SYSTEM TestDataType
  (* Version 1.0, 2024-01-14, ADMIN *)
  APPLICATION TestDataTypeApp
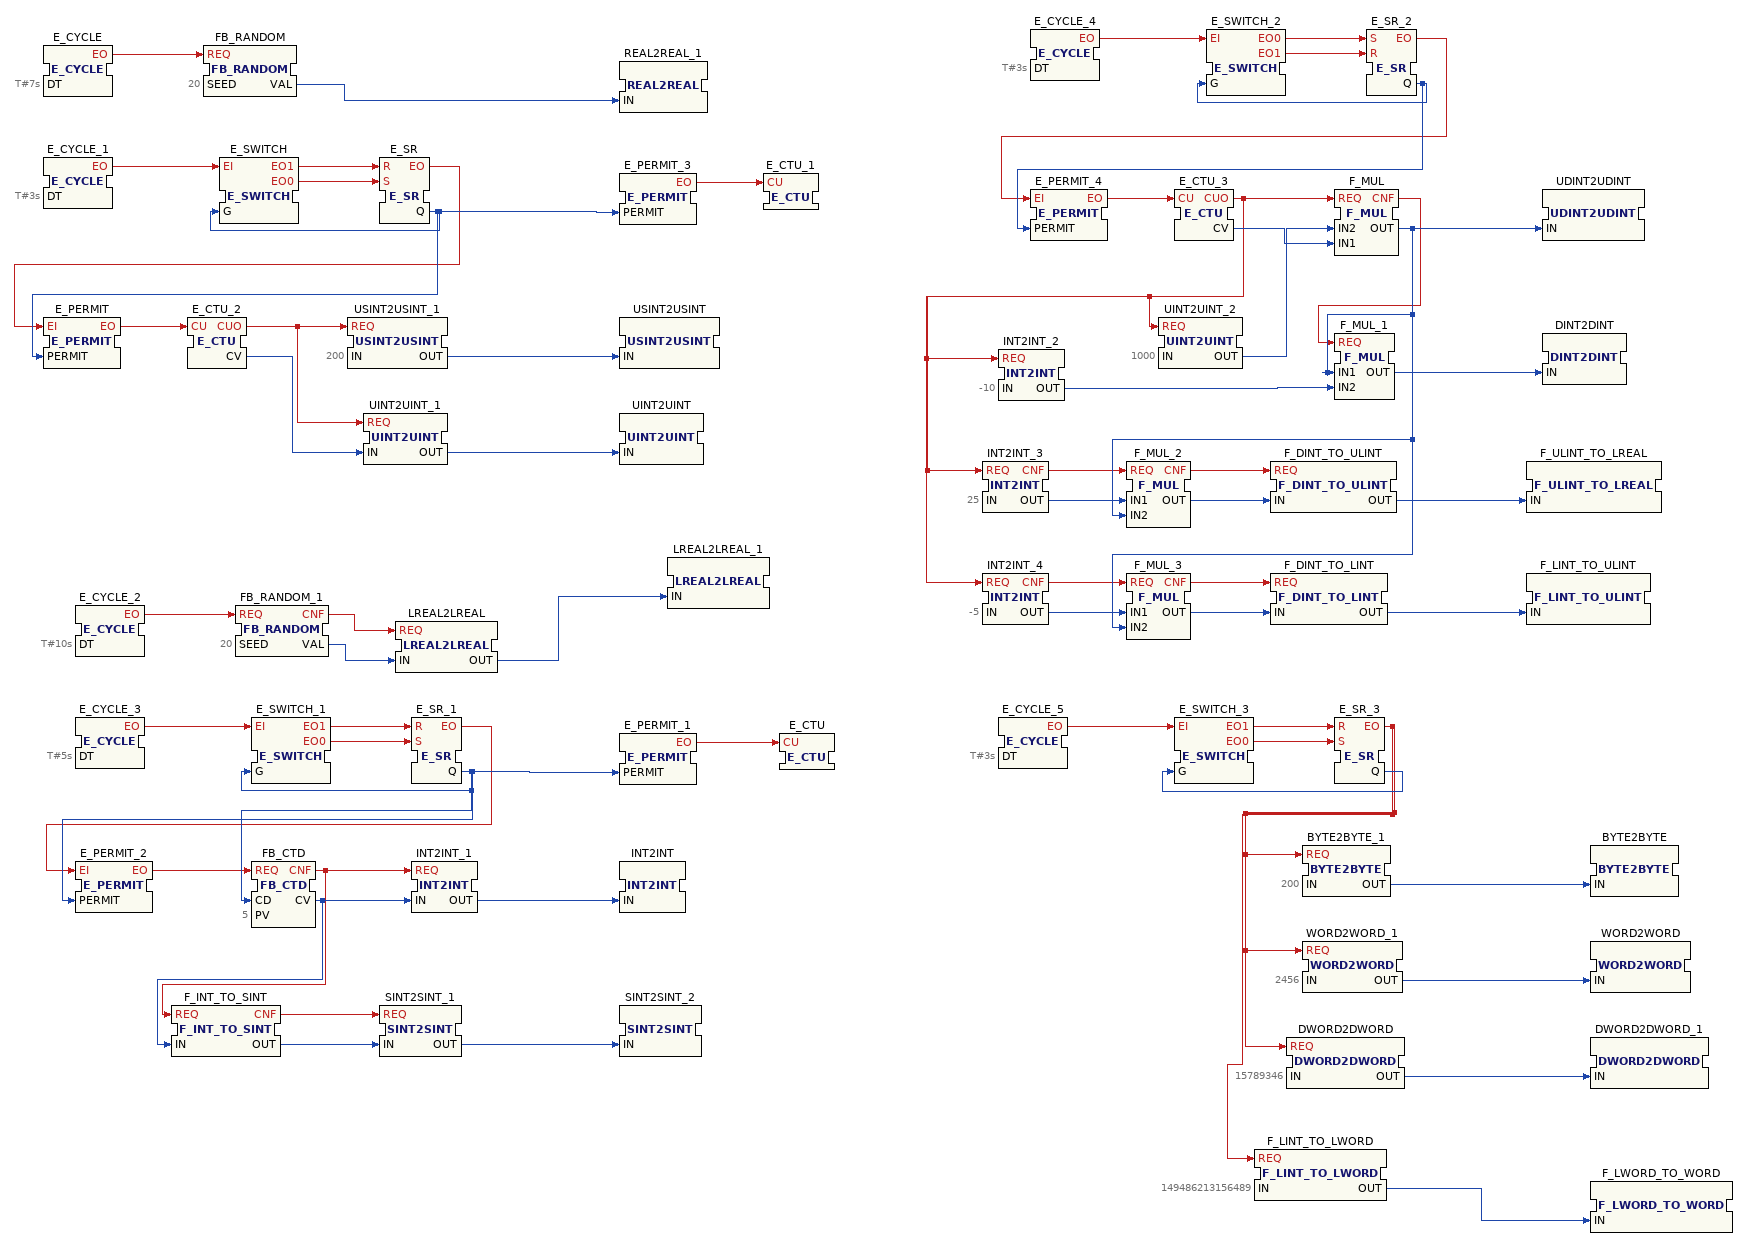
    FBS
      E_CYCLE : E_CYCLE(DT := T#7s);
      FB_RANDOM : FB_RANDOM(SEED := 20);
      E_CYCLE_1 : E_CYCLE(DT := T#3s);
      E_SWITCH : E_SWITCH;
      E_SR : E_SR;
      E_PERMIT : E_PERMIT;
      E_PERMIT_1 : E_PERMIT;
      E_CTU : E_CTU;
      E_CYCLE_2 : E_CYCLE(DT := T#10s);
      FB_RANDOM_1 : FB_RANDOM(SEED := 20);
      E_CYCLE_3 : E_CYCLE(DT := T#5s);
      E_SWITCH_1 : E_SWITCH;
      E_SR_1 : E_SR;
      E_PERMIT_2 : E_PERMIT;
      REAL2REAL_1 : REAL2REAL;
      E_PERMIT_3 : E_PERMIT;
      E_CTU_1 : E_CTU;
      UINT2UINT : UINT2UINT;
      INT2INT : INT2INT;
      SINT2SINT_1 : SINT2SINT;
      USINT2USINT : USINT2USINT;
      E_CTU_2 : E_CTU;
      UINT2UINT_1 : UINT2UINT;
      SINT2SINT_2 : SINT2SINT;
      INT2INT_1 : INT2INT;
      USINT2USINT_1 : USINT2USINT(IN := 200);
      LREAL2LREAL : LREAL2LREAL;
      LREAL2LREAL_1 : LREAL2LREAL;
      UDINT2UDINT : UDINT2UDINT;
      DINT2DINT : DINT2DINT;
      F_MUL : F_MUL;
      UINT2UINT_2 : UINT2UINT(IN := 1000);
      FB_CTD : FB_CTD(PV := 5);
      F_INT_TO_SINT : F_INT_TO_SINT;
      E_CYCLE_4 : E_CYCLE(DT := T#3s);
      E_SWITCH_2 : E_SWITCH;
      E_SR_2 : E_SR;
      E_PERMIT_4 : E_PERMIT;
      E_CTU_3 : E_CTU;
      F_MUL_1 : F_MUL;
      INT2INT_2 : INT2INT(IN := -10);
      BYTE2BYTE : BYTE2BYTE;
      WORD2WORD : WORD2WORD;
      F_DINT_TO_LINT : F_DINT_TO_LINT;
      F_LINT_TO_ULINT : F_LINT_TO_ULINT;
      F_DINT_TO_ULINT : F_DINT_TO_ULINT;
      INT2INT_3 : INT2INT(IN := 25);
      F_MUL_2 : F_MUL;
      F_ULINT_TO_LREAL : F_ULINT_TO_LREAL;
      INT2INT_4 : INT2INT(IN := -5);
      F_MUL_3 : F_MUL;
      E_SWITCH_3 : E_SWITCH;
      E_SR_3 : E_SR;
      E_CYCLE_5 : E_CYCLE(DT := T#3s);
      BYTE2BYTE_1 : BYTE2BYTE(IN := 200);
      DWORD2DWORD : DWORD2DWORD(IN := 15789346);
      WORD2WORD_1 : WORD2WORD(IN := 2456);
      DWORD2DWORD_1 : DWORD2DWORD;
      F_LWORD_TO_WORD : F_LWORD_TO_WORD;
      F_LINT_TO_LWORD : F_LINT_TO_LWORD(IN := 149486213156489);
    END_FBS
    EVENT_CONNECTIONS
      E_CYCLE.EO TO FB_RANDOM.REQ;
      E_SWITCH.EO1 TO E_SR.R;
      E_SWITCH.EO0 TO E_SR.S;
      E_SR.EO TO E_PERMIT.EI;
      E_CYCLE_1.EO TO E_SWITCH.EI;
      E_PERMIT_1.EO TO E_CTU.CU;
      E_PERMIT_3.EO TO E_CTU_1.CU;
      E_SR_1.EO TO E_PERMIT_2.EI;
      E_CYCLE_2.EO TO FB_RANDOM_1.REQ;
      E_SWITCH_1.EO1 TO E_SR_1.R;
      E_CYCLE_3.EO TO E_SWITCH_1.EI;
      E_SWITCH_1.EO0 TO E_SR_1.S;
      E_PERMIT.EO TO E_CTU_2.CU;
      E_CTU_2.CUO TO UINT2UINT_1.REQ;
      E_CTU_2.CUO TO USINT2USINT_1.REQ;
      FB_RANDOM_1.CNF TO LREAL2LREAL.REQ;
      E_PERMIT_2.EO TO FB_CTD.REQ;
      FB_CTD.CNF TO INT2INT_1.REQ;
      F_INT_TO_SINT.CNF TO SINT2SINT_1.REQ;
      FB_CTD.CNF TO F_INT_TO_SINT.REQ;
      E_PERMIT_4.EO TO E_CTU_3.CU;
      E_CYCLE_4.EO TO E_SWITCH_2.EI;
      E_SWITCH_2.EO0 TO E_SR_2.S;
      E_SR_2.EO TO E_PERMIT_4.EI;
      E_SWITCH_2.EO1 TO E_SR_2.R;
      E_CTU_3.CUO TO F_MUL.REQ;
      E_CTU_3.CUO TO UINT2UINT_2.REQ;
      E_CTU_3.CUO TO INT2INT_2.REQ;
      F_MUL.CNF TO F_MUL_1.REQ;
      E_CTU_3.CUO TO INT2INT_3.REQ;
      INT2INT_3.CNF TO F_MUL_2.REQ;
      F_MUL_2.CNF TO F_DINT_TO_ULINT.REQ;
      F_MUL_3.CNF TO F_DINT_TO_LINT.REQ;
      E_CTU_3.CUO TO INT2INT_4.REQ;
      INT2INT_4.CNF TO F_MUL_3.REQ;
      E_CYCLE_5.EO TO E_SWITCH_3.EI;
      E_SWITCH_3.EO1 TO E_SR_3.R;
      E_SWITCH_3.EO0 TO E_SR_3.S;
      E_SR_3.EO TO BYTE2BYTE_1.REQ;
      E_SR_3.EO TO WORD2WORD_1.REQ;
      E_SR_3.EO TO DWORD2DWORD.REQ;
      E_SR_3.EO TO F_LINT_TO_LWORD.REQ;
    END_CONNECTIONS
    DATA_CONNECTIONS
      E_SR.Q TO E_SWITCH.G;
      E_SR.Q TO E_PERMIT.PERMIT;
      E_SR_1.Q TO E_SWITCH_1.G;
      E_SR_1.Q TO E_PERMIT_2.PERMIT;
      E_SR.Q TO E_PERMIT_3.PERMIT;
      E_SR_1.Q TO E_PERMIT_1.PERMIT;
      FB_RANDOM.VAL TO REAL2REAL_1.IN;
      E_CTU_2.CV TO UINT2UINT_1.IN;
      INT2INT_1.OUT TO INT2INT.IN;
      SINT2SINT_1.OUT TO SINT2SINT_2.IN;
      USINT2USINT_1.OUT TO USINT2USINT.IN;
      UINT2UINT_1.OUT TO UINT2UINT.IN;
      FB_RANDOM_1.VAL TO LREAL2LREAL.IN;
      LREAL2LREAL.OUT TO LREAL2LREAL_1.IN;
      FB_CTD.CV TO INT2INT_1.IN;
      F_INT_TO_SINT.OUT TO SINT2SINT_1.IN;
      FB_CTD.CV TO F_INT_TO_SINT.IN;
      E_SR_2.Q TO E_PERMIT_4.PERMIT;
      E_SR_2.Q TO E_SWITCH_2.G;
      UINT2UINT_2.OUT TO F_MUL.IN2;
      E_CTU_3.CV TO F_MUL.IN1;
      F_MUL.OUT TO F_MUL_1.IN1;
      INT2INT_2.OUT TO F_MUL_1.IN2;
      F_MUL.OUT TO UDINT2UDINT.IN;
      F_MUL_1.OUT TO DINT2DINT.IN;
      E_SR_1.Q TO FB_CTD.CD;
      INT2INT_3.OUT TO F_MUL_2.IN1;
      F_MUL.OUT TO F_MUL_2.IN2;
      F_MUL_2.OUT TO F_DINT_TO_ULINT.IN;
      F_DINT_TO_LINT.OUT TO F_LINT_TO_ULINT.IN;
      F_DINT_TO_ULINT.OUT TO F_ULINT_TO_LREAL.IN;
      INT2INT_4.OUT TO F_MUL_3.IN1;
      F_MUL.OUT TO F_MUL_3.IN2;
      F_MUL_3.OUT TO F_DINT_TO_LINT.IN;
      E_SR_3.Q TO E_SWITCH_3.G;
      BYTE2BYTE_1.OUT TO BYTE2BYTE.IN;
      WORD2WORD_1.OUT TO WORD2WORD.IN;
      DWORD2DWORD.OUT TO DWORD2DWORD_1.IN;
      F_LINT_TO_LWORD.OUT TO F_LWORD_TO_WORD.IN;
    END_CONNECTIONS
  END_APPLICATION
  DEVICE BeagleBoneBlack : BeagleBoneBlack(MGR_ID := "localhost:61500")
    {SET_ATTRIBUTE(Profile, HOLOBLOC)} (* device profile *)
    RESOURCE EMB_RES : EMB_RES
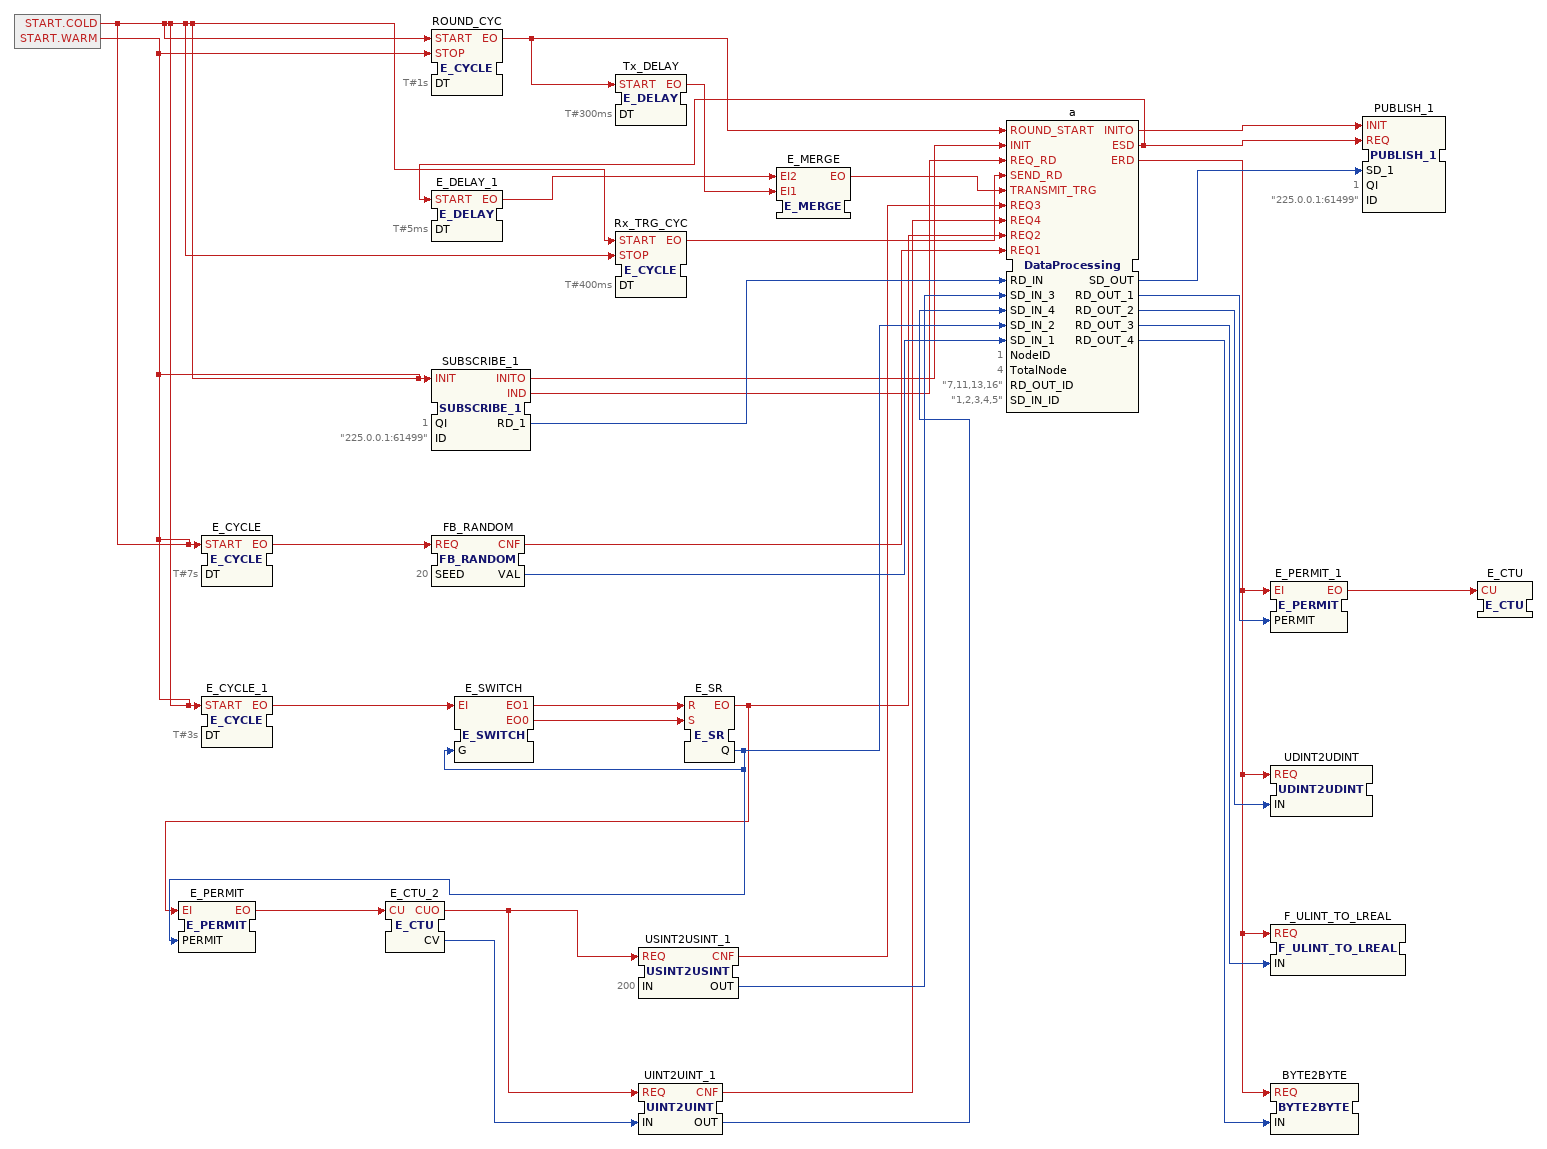
      FBS
        a : DataProcessing(NodeID := 1, TotalNode := 4, RD_OUT_ID := "7,11,13,16", SD_IN_ID := "1,2,3,4,5");
        Rx_TRG_CYC : E_CYCLE(DT := T#400ms);
        PUBLISH_1 : PUBLISH_1(QI := 1, ID := "225.0.0.1:61499");
        E_DELAY_1 : E_DELAY(DT := T#5ms);
        SUBSCRIBE_1 : SUBSCRIBE_1(QI := 1, ID := "225.0.0.1:61499");
        E_MERGE : E_MERGE;
        Tx_DELAY : E_DELAY(DT := T#300ms);
        ROUND_CYC : E_CYCLE(DT := T#1s);
        F_ULINT_TO_LREAL : F_ULINT_TO_LREAL;
        BYTE2BYTE : BYTE2BYTE;
        UDINT2UDINT : UDINT2UDINT;
        USINT2USINT_1 : USINT2USINT(IN := 200);
        UINT2UINT_1 : UINT2UINT;
        E_CTU_2 : E_CTU;
        E_CTU : E_CTU;
        E_PERMIT_1 : E_PERMIT;
        E_PERMIT : E_PERMIT;
        E_SR : E_SR;
        E_SWITCH : E_SWITCH;
        E_CYCLE_1 : E_CYCLE(DT := T#3s);
        FB_RANDOM : FB_RANDOM(SEED := 20);
        E_CYCLE : E_CYCLE(DT := T#7s);
      END_FBS
      EVENT_CONNECTIONS
        ROUND_CYC.EO TO a.ROUND_START;
        ROUND_CYC.EO TO Tx_DELAY.START;
        SUBSCRIBE_1.INITO TO a.INIT;
        SUBSCRIBE_1.IND TO a.REQ_RD;
        a.INITO TO PUBLISH_1.INIT;
        E_DELAY_1.EO TO E_MERGE.EI2;
        Tx_DELAY.EO TO E_MERGE.EI1;
        START.COLD TO ROUND_CYC.START;
        START.WARM TO ROUND_CYC.STOP;
        START.COLD TO Rx_TRG_CYC.START;
        START.COLD TO Rx_TRG_CYC.STOP;
        START.COLD TO SUBSCRIBE_1.INIT;
        START.WARM TO SUBSCRIBE_1.INIT;
        a.ESD TO PUBLISH_1.REQ;
        a.ESD TO E_DELAY_1.START;
        Rx_TRG_CYC.EO TO a.SEND_RD;
        E_MERGE.EO TO a.TRANSMIT_TRG;
        a.ERD TO F_ULINT_TO_LREAL.REQ;
        a.ERD TO UDINT2UDINT.REQ;
        USINT2USINT_1.CNF TO a.REQ3;
        UINT2UINT_1.CNF TO a.REQ4;
        E_CTU_2.CUO TO UINT2UINT_1.REQ;
        E_CTU_2.CUO TO USINT2USINT_1.REQ;
        E_PERMIT_1.EO TO E_CTU.CU;
        a.ERD TO E_PERMIT_1.EI;
        E_PERMIT.EO TO E_CTU_2.CU;
        E_SR.EO TO E_PERMIT.EI;
        E_SR.EO TO a.REQ2;
        E_SWITCH.EO1 TO E_SR.R;
        E_SWITCH.EO0 TO E_SR.S;
        E_CYCLE_1.EO TO E_SWITCH.EI;
        START.COLD TO E_CYCLE_1.START;
        START.WARM TO E_CYCLE_1.START;
        FB_RANDOM.CNF TO a.REQ1;
        E_CYCLE.EO TO FB_RANDOM.REQ;
        START.COLD TO E_CYCLE.START;
        START.WARM TO E_CYCLE.START;
        a.ERD TO BYTE2BYTE.REQ;
      END_CONNECTIONS
      DATA_CONNECTIONS
        SUBSCRIBE_1.RD_1 TO a.RD_IN;
        a.SD_OUT TO PUBLISH_1.SD_1;
        USINT2USINT_1.OUT TO a.SD_IN_3;
        UINT2UINT_1.OUT TO a.SD_IN_4;
        E_CTU_2.CV TO UINT2UINT_1.IN;
        E_SR.Q TO E_PERMIT.PERMIT;
        E_SR.Q TO a.SD_IN_2;
        E_SR.Q TO E_SWITCH.G;
        FB_RANDOM.VAL TO a.SD_IN_1;
        a.RD_OUT_1 TO E_PERMIT_1.PERMIT;
        a.RD_OUT_2 TO UDINT2UDINT.IN;
        a.RD_OUT_3 TO F_ULINT_TO_LREAL.IN;
        a.RD_OUT_4 TO BYTE2BYTE.IN;
      END_CONNECTIONS
    END_RESOURCE
  END_DEVICE
  DEVICE BeagleBoneBlack_1 : BeagleBoneBlack(MGR_ID := "localhost:61501")
    {SET_ATTRIBUTE(Profile, HOLOBLOC)} (* device profile *)
    RESOURCE EMB_RES : EMB_RES
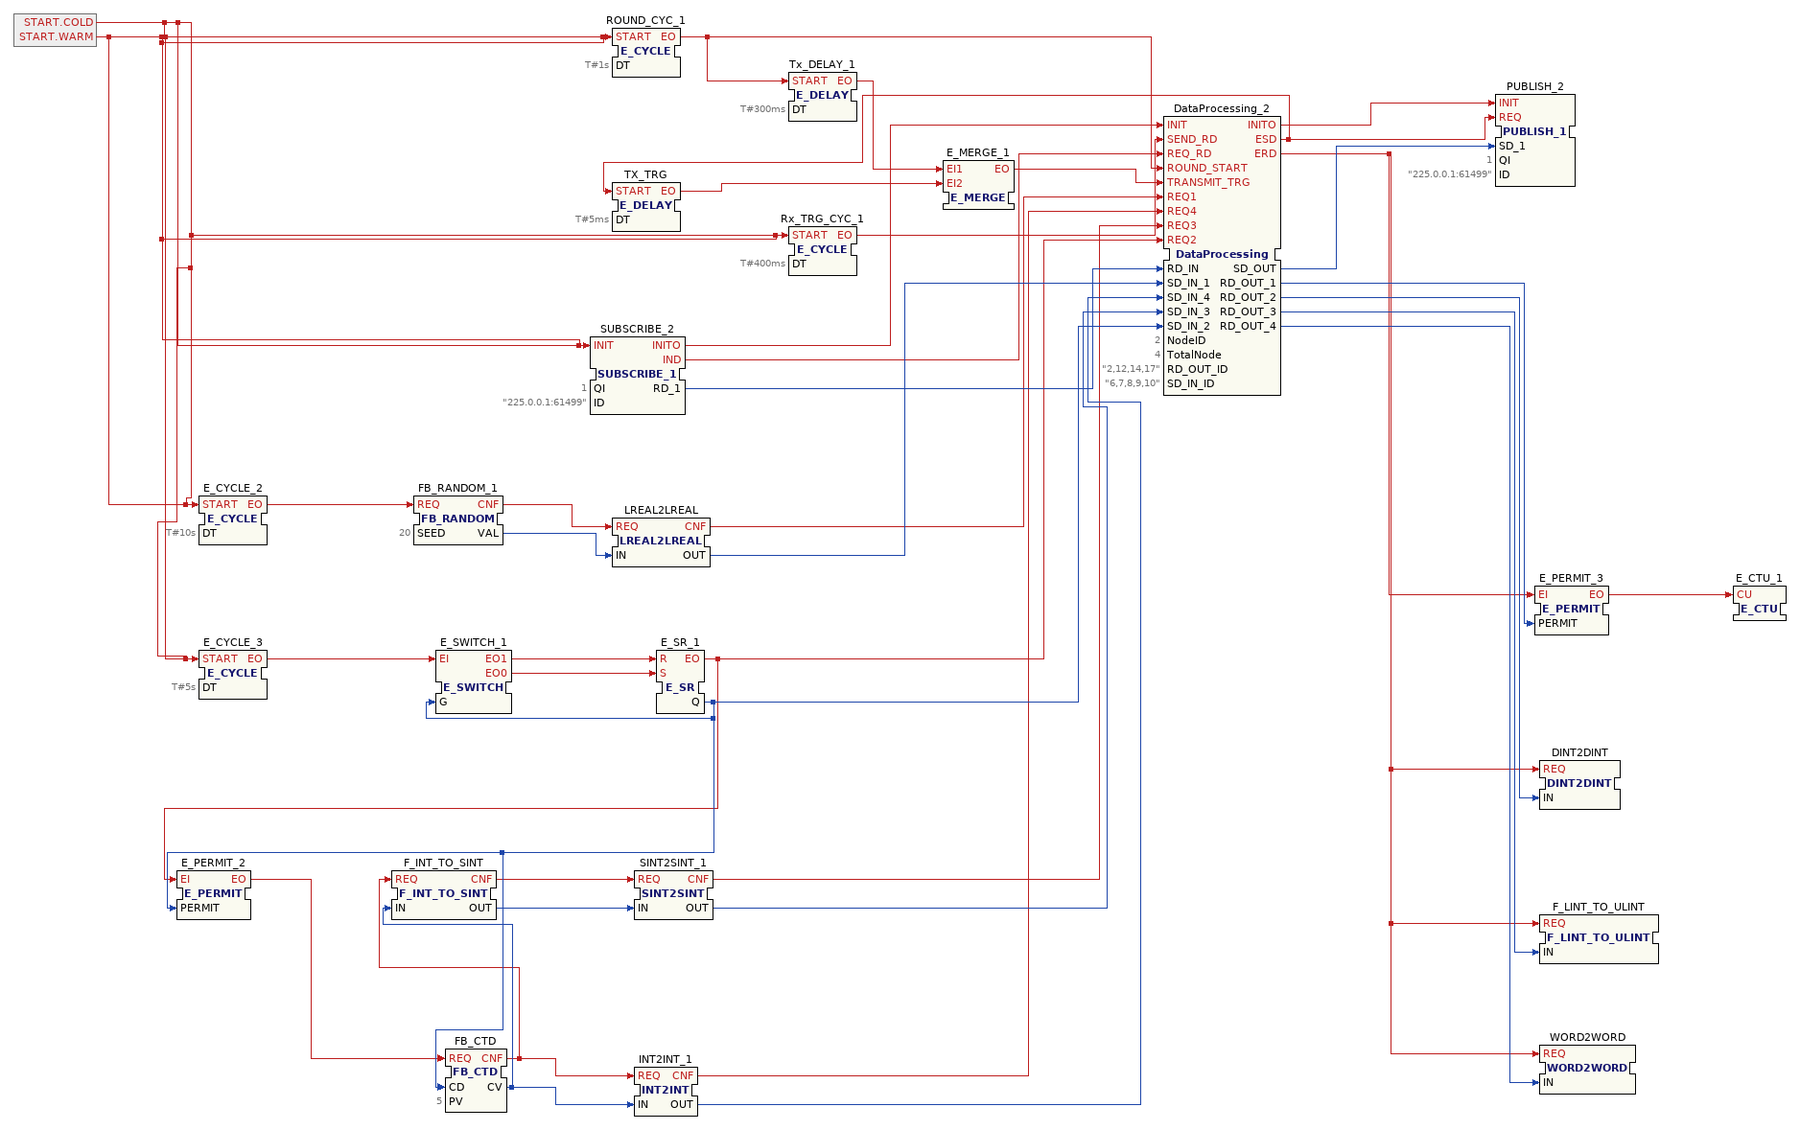
      FBS
        E_MERGE_1 : E_MERGE;
        Tx_DELAY_1 : E_DELAY(DT := T#300ms);
        TX_TRG : E_DELAY(DT := T#5ms);
        PUBLISH_2 : PUBLISH_1(QI := 1, ID := "225.0.0.1:61499");
        SUBSCRIBE_2 : SUBSCRIBE_1(QI := 1, ID := "225.0.0.1:61499");
        DataProcessing_2 : DataProcessing(NodeID := 2, TotalNode := 4, RD_OUT_ID := "2,12,14,17", SD_IN_ID := "6,7,8,9,10");
        Rx_TRG_CYC_1 : E_CYCLE(DT := T#400ms);
        ROUND_CYC_1 : E_CYCLE(DT := T#1s);
        F_LINT_TO_ULINT : F_LINT_TO_ULINT;
        WORD2WORD : WORD2WORD;
        F_INT_TO_SINT : F_INT_TO_SINT;
        FB_CTD : FB_CTD(PV := 5);
        DINT2DINT : DINT2DINT;
        LREAL2LREAL : LREAL2LREAL;
        INT2INT_1 : INT2INT;
        SINT2SINT_1 : SINT2SINT;
        E_CTU_1 : E_CTU;
        E_PERMIT_3 : E_PERMIT;
        E_PERMIT_2 : E_PERMIT;
        E_SR_1 : E_SR;
        E_SWITCH_1 : E_SWITCH;
        E_CYCLE_3 : E_CYCLE(DT := T#5s);
        FB_RANDOM_1 : FB_RANDOM(SEED := 20);
        E_CYCLE_2 : E_CYCLE(DT := T#10s);
      END_FBS
      EVENT_CONNECTIONS
        SUBSCRIBE_2.INITO TO DataProcessing_2.INIT;
        Tx_DELAY_1.EO TO E_MERGE_1.EI1;
        ROUND_CYC_1.EO TO Tx_DELAY_1.START;
        DataProcessing_2.INITO TO PUBLISH_2.INIT;
        TX_TRG.EO TO E_MERGE_1.EI2;
        Rx_TRG_CYC_1.EO TO DataProcessing_2.SEND_RD;
        SUBSCRIBE_2.IND TO DataProcessing_2.REQ_RD;
        ROUND_CYC_1.EO TO DataProcessing_2.ROUND_START;
        START.COLD TO ROUND_CYC_1.START;
        START.WARM TO ROUND_CYC_1.START;
        START.COLD TO SUBSCRIBE_2.INIT;
        START.WARM TO SUBSCRIBE_2.INIT;
        START.COLD TO Rx_TRG_CYC_1.START;
        START.WARM TO Rx_TRG_CYC_1.START;
        DataProcessing_2.ESD TO PUBLISH_2.REQ;
        DataProcessing_2.ESD TO TX_TRG.START;
        E_MERGE_1.EO TO DataProcessing_2.TRANSMIT_TRG;
        DataProcessing_2.ERD TO F_LINT_TO_ULINT.REQ;
        FB_CTD.CNF TO F_INT_TO_SINT.REQ;
        DataProcessing_2.ERD TO DINT2DINT.REQ;
        LREAL2LREAL.CNF TO DataProcessing_2.REQ1;
        INT2INT_1.CNF TO DataProcessing_2.REQ4;
        FB_CTD.CNF TO INT2INT_1.REQ;
        SINT2SINT_1.CNF TO DataProcessing_2.REQ3;
        F_INT_TO_SINT.CNF TO SINT2SINT_1.REQ;
        E_PERMIT_3.EO TO E_CTU_1.CU;
        DataProcessing_2.ERD TO E_PERMIT_3.EI;
        E_PERMIT_2.EO TO FB_CTD.REQ;
        E_SR_1.EO TO DataProcessing_2.REQ2;
        E_SR_1.EO TO E_PERMIT_2.EI;
        E_SWITCH_1.EO1 TO E_SR_1.R;
        E_SWITCH_1.EO0 TO E_SR_1.S;
        E_CYCLE_3.EO TO E_SWITCH_1.EI;
        START.WARM TO E_CYCLE_3.START;
        START.COLD TO E_CYCLE_3.START;
        FB_RANDOM_1.CNF TO LREAL2LREAL.REQ;
        E_CYCLE_2.EO TO FB_RANDOM_1.REQ;
        START.WARM TO E_CYCLE_2.START;
        START.COLD TO E_CYCLE_2.START;
        DataProcessing_2.ERD TO WORD2WORD.REQ;
      END_CONNECTIONS
      DATA_CONNECTIONS
        SUBSCRIBE_2.RD_1 TO DataProcessing_2.RD_IN;
        DataProcessing_2.SD_OUT TO PUBLISH_2.SD_1;
        FB_CTD.CV TO F_INT_TO_SINT.IN;
        LREAL2LREAL.OUT TO DataProcessing_2.SD_IN_1;
        INT2INT_1.OUT TO DataProcessing_2.SD_IN_4;
        FB_CTD.CV TO INT2INT_1.IN;
        SINT2SINT_1.OUT TO DataProcessing_2.SD_IN_3;
        F_INT_TO_SINT.OUT TO SINT2SINT_1.IN;
        E_SR_1.Q TO DataProcessing_2.SD_IN_2;
        E_SR_1.Q TO E_PERMIT_2.PERMIT;
        E_SR_1.Q TO FB_CTD.CD;
        E_SR_1.Q TO E_SWITCH_1.G;
        FB_RANDOM_1.VAL TO LREAL2LREAL.IN;
        DataProcessing_2.RD_OUT_1 TO E_PERMIT_3.PERMIT;
        DataProcessing_2.RD_OUT_2 TO DINT2DINT.IN;
        DataProcessing_2.RD_OUT_3 TO F_LINT_TO_ULINT.IN;
        DataProcessing_2.RD_OUT_4 TO WORD2WORD.IN;
      END_CONNECTIONS
    END_RESOURCE
  END_DEVICE
  DEVICE BeagleBoneBlack_2 : BeagleBoneBlack(MGR_ID := "localhost:61502")
    {SET_ATTRIBUTE(Profile, HOLOBLOC)} (* device profile *)
    RESOURCE EMB_RES : EMB_RES
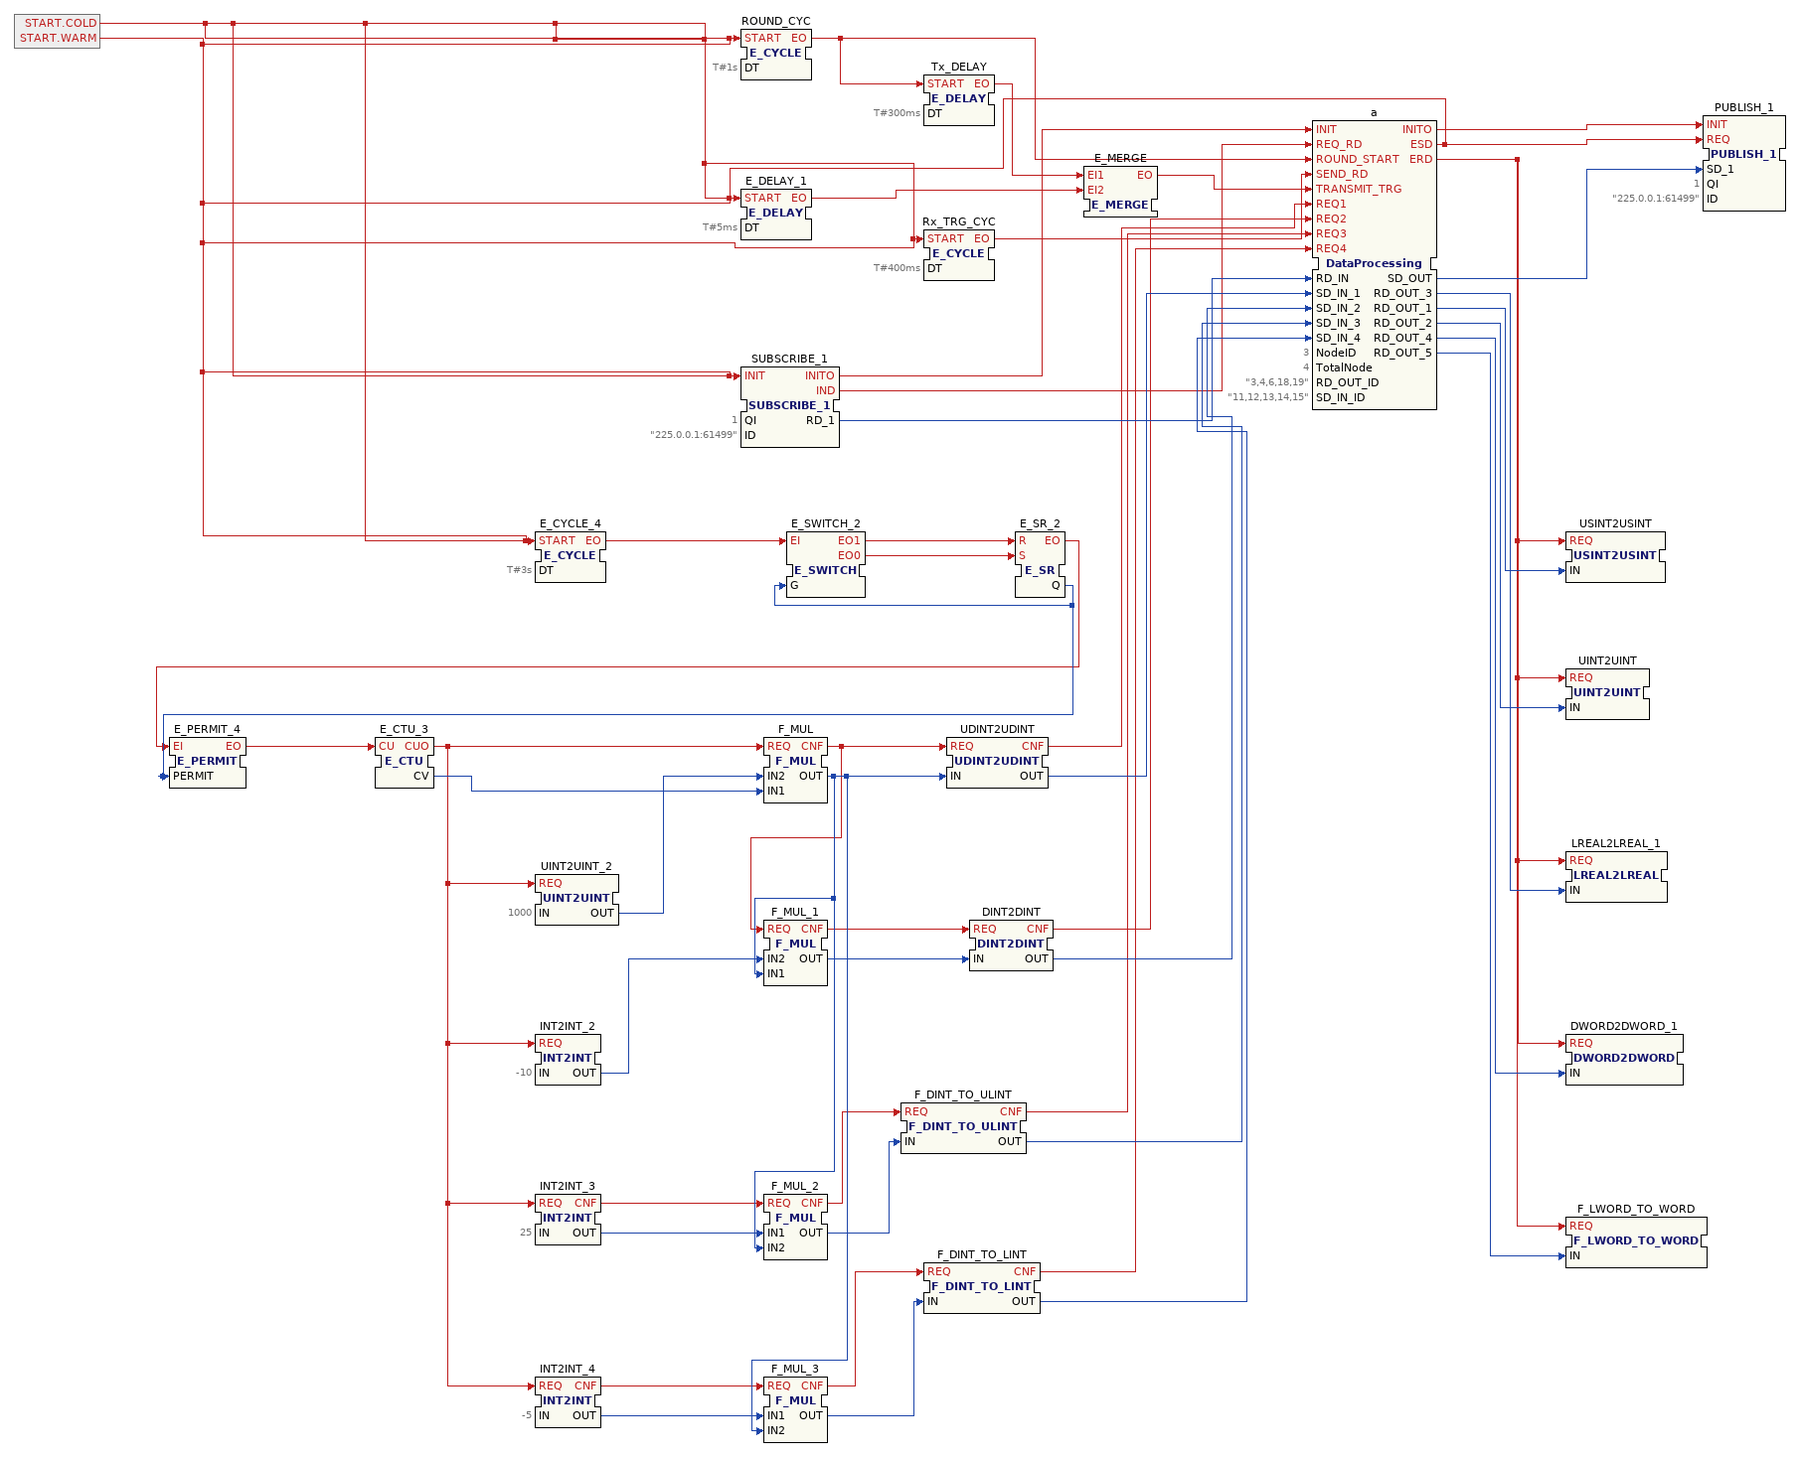
      FBS
        SUBSCRIBE_1 : SUBSCRIBE_1(QI := 1, ID := "225.0.0.1:61499");
        ROUND_CYC : E_CYCLE(DT := T#1s);
        E_MERGE : E_MERGE;
        E_DELAY_1 : E_DELAY(DT := T#5ms);
        Rx_TRG_CYC : E_CYCLE(DT := T#400ms);
        PUBLISH_1 : PUBLISH_1(QI := 1, ID := "225.0.0.1:61499");
        Tx_DELAY : E_DELAY(DT := T#300ms);
        a : DataProcessing(NodeID := 3, TotalNode := 4, RD_OUT_ID := "3,4,6,18,19", SD_IN_ID := "11,12,13,14,15");
        UDINT2UDINT : UDINT2UDINT;
        DINT2DINT : DINT2DINT;
        F_MUL_3 : F_MUL;
        INT2INT_4 : INT2INT(IN := -5);
        F_MUL_2 : F_MUL;
        INT2INT_3 : INT2INT(IN := 25);
        F_DINT_TO_ULINT : F_DINT_TO_ULINT;
        F_DINT_TO_LINT : F_DINT_TO_LINT;
        INT2INT_2 : INT2INT(IN := -10);
        F_MUL_1 : F_MUL;
        E_CTU_3 : E_CTU;
        E_PERMIT_4 : E_PERMIT;
        E_SR_2 : E_SR;
        E_SWITCH_2 : E_SWITCH;
        E_CYCLE_4 : E_CYCLE(DT := T#3s);
        UINT2UINT_2 : UINT2UINT(IN := 1000);
        F_MUL : F_MUL;
        LREAL2LREAL_1 : LREAL2LREAL;
        USINT2USINT : USINT2USINT;
        UINT2UINT : UINT2UINT;
        DWORD2DWORD_1 : DWORD2DWORD;
        F_LWORD_TO_WORD : F_LWORD_TO_WORD;
      END_FBS
      EVENT_CONNECTIONS
        SUBSCRIBE_1.INITO TO a.INIT;
        SUBSCRIBE_1.IND TO a.REQ_RD;
        a.INITO TO PUBLISH_1.INIT;
        ROUND_CYC.EO TO a.ROUND_START;
        a.ESD TO E_DELAY_1.START;
        Rx_TRG_CYC.EO TO a.SEND_RD;
        E_MERGE.EO TO a.TRANSMIT_TRG;
        Tx_DELAY.EO TO E_MERGE.EI1;
        ROUND_CYC.EO TO Tx_DELAY.START;
        a.ESD TO PUBLISH_1.REQ;
        E_DELAY_1.EO TO E_MERGE.EI2;
        UDINT2UDINT.CNF TO a.REQ1;
        DINT2DINT.CNF TO a.REQ2;
        START.COLD TO ROUND_CYC.START;
        START.WARM TO ROUND_CYC.START;
        START.COLD TO E_DELAY_1.START;
        START.WARM TO E_DELAY_1.START;
        START.COLD TO SUBSCRIBE_1.INIT;
        START.WARM TO SUBSCRIBE_1.INIT;
        START.COLD TO Rx_TRG_CYC.START;
        START.WARM TO Rx_TRG_CYC.START;
        INT2INT_4.CNF TO F_MUL_3.REQ;
        INT2INT_3.CNF TO F_MUL_2.REQ;
        F_DINT_TO_ULINT.CNF TO a.REQ3;
        F_MUL_2.CNF TO F_DINT_TO_ULINT.REQ;
        F_DINT_TO_LINT.CNF TO a.REQ4;
        F_MUL_3.CNF TO F_DINT_TO_LINT.REQ;
        F_MUL_1.CNF TO DINT2DINT.REQ;
        E_CTU_3.CUO TO INT2INT_2.REQ;
        E_CTU_3.CUO TO INT2INT_3.REQ;
        E_CTU_3.CUO TO INT2INT_4.REQ;
        E_PERMIT_4.EO TO E_CTU_3.CU;
        E_SR_2.EO TO E_PERMIT_4.EI;
        E_SWITCH_2.EO1 TO E_SR_2.R;
        E_SWITCH_2.EO0 TO E_SR_2.S;
        E_CYCLE_4.EO TO E_SWITCH_2.EI;
        START.COLD TO E_CYCLE_4.START;
        START.WARM TO E_CYCLE_4.START;
        E_CTU_3.CUO TO UINT2UINT_2.REQ;
        F_MUL.CNF TO UDINT2UDINT.REQ;
        F_MUL.CNF TO F_MUL_1.REQ;
        E_CTU_3.CUO TO F_MUL.REQ;
        a.ERD TO LREAL2LREAL_1.REQ;
        a.ERD TO USINT2USINT.REQ;
        a.ERD TO UINT2UINT.REQ;
        a.ERD TO DWORD2DWORD_1.REQ;
        a.ERD TO F_LWORD_TO_WORD.REQ;
      END_CONNECTIONS
      DATA_CONNECTIONS
        a.SD_OUT TO PUBLISH_1.SD_1;
        SUBSCRIBE_1.RD_1 TO a.RD_IN;
        UDINT2UDINT.OUT TO a.SD_IN_1;
        DINT2DINT.OUT TO a.SD_IN_2;
        INT2INT_4.OUT TO F_MUL_3.IN1;
        INT2INT_3.OUT TO F_MUL_2.IN1;
        F_DINT_TO_ULINT.OUT TO a.SD_IN_3;
        F_MUL_2.OUT TO F_DINT_TO_ULINT.IN;
        F_DINT_TO_LINT.OUT TO a.SD_IN_4;
        F_MUL_3.OUT TO F_DINT_TO_LINT.IN;
        F_MUL_1.OUT TO DINT2DINT.IN;
        INT2INT_2.OUT TO F_MUL_1.IN2;
        E_SR_2.Q TO E_PERMIT_4.PERMIT;
        E_SR_2.Q TO E_SWITCH_2.G;
        F_MUL.OUT TO F_MUL_1.IN1;
        F_MUL.OUT TO UDINT2UDINT.IN;
        F_MUL.OUT TO F_MUL_2.IN2;
        F_MUL.OUT TO F_MUL_3.IN2;
        UINT2UINT_2.OUT TO F_MUL.IN2;
        E_CTU_3.CV TO F_MUL.IN1;
        a.RD_OUT_3 TO LREAL2LREAL_1.IN;
        a.RD_OUT_1 TO USINT2USINT.IN;
        a.RD_OUT_2 TO UINT2UINT.IN;
        a.RD_OUT_4 TO DWORD2DWORD_1.IN;
        a.RD_OUT_5 TO F_LWORD_TO_WORD.IN;
      END_CONNECTIONS
    END_RESOURCE
  END_DEVICE
  DEVICE BeagleBoneBlack_3 : BeagleBoneBlack(MGR_ID := "localhost:61503")
    {SET_ATTRIBUTE(Profile, HOLOBLOC)} (* device profile *)
    RESOURCE EMB_RES : EMB_RES
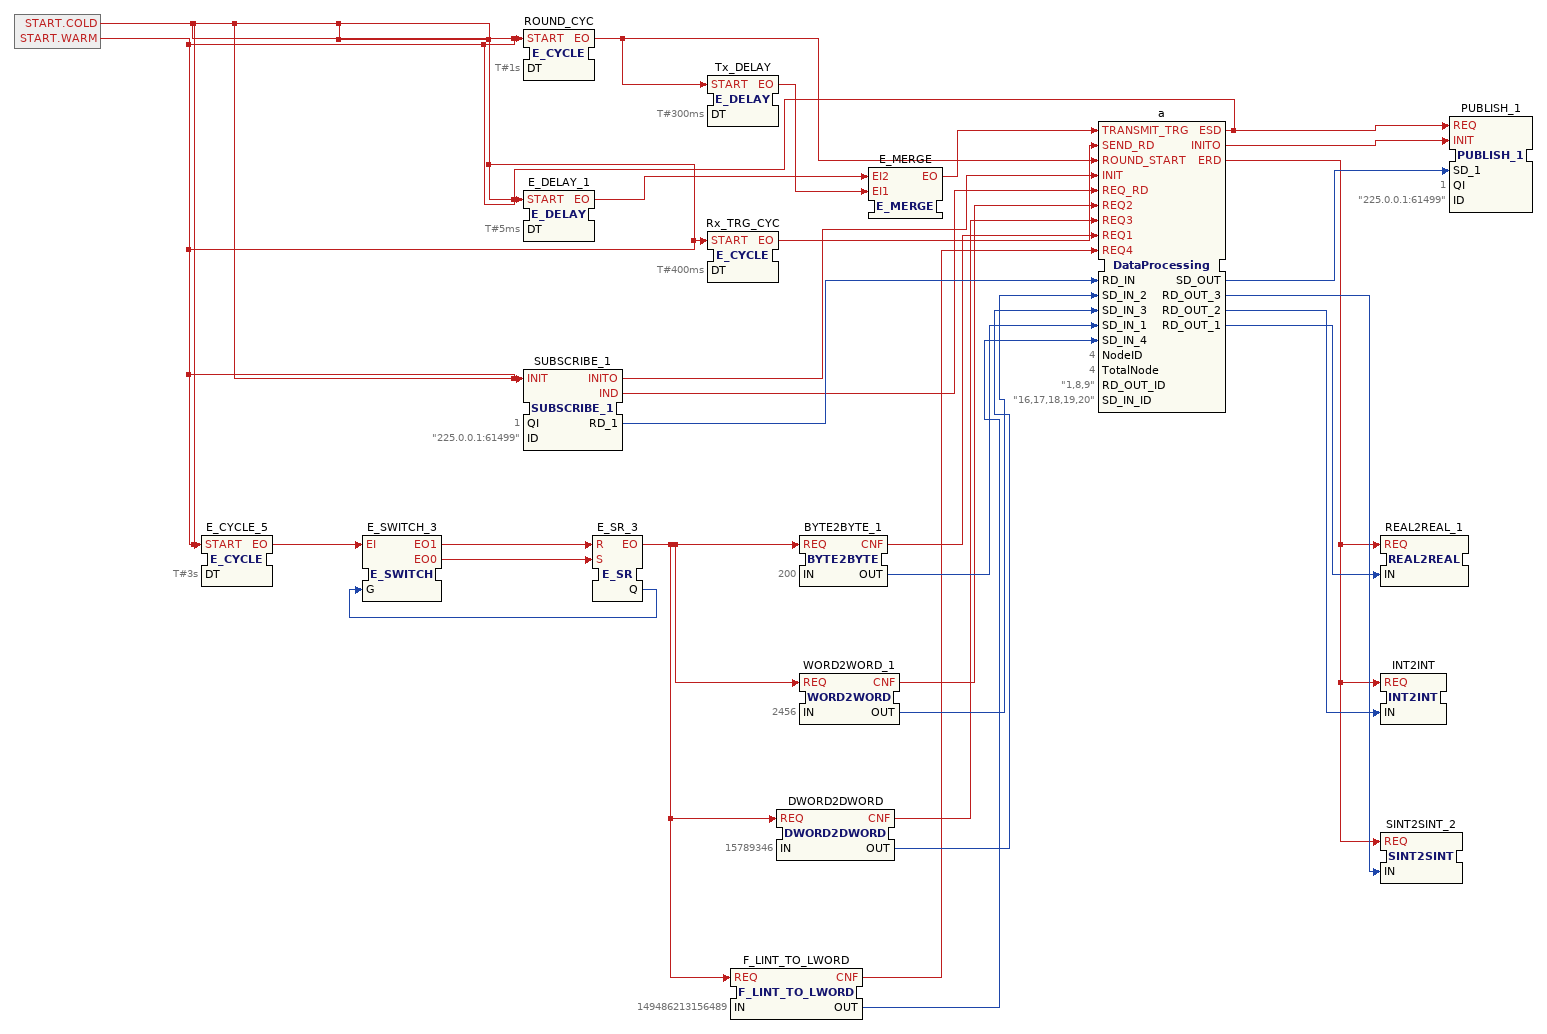
      FBS
        Rx_TRG_CYC : E_CYCLE(DT := T#400ms);
        Tx_DELAY : E_DELAY(DT := T#300ms);
        PUBLISH_1 : PUBLISH_1(QI := 1, ID := "225.0.0.1:61499");
        E_DELAY_1 : E_DELAY(DT := T#5ms);
        ROUND_CYC : E_CYCLE(DT := T#1s);
        SUBSCRIBE_1 : SUBSCRIBE_1(QI := 1, ID := "225.0.0.1:61499");
        a : DataProcessing(NodeID := 4, TotalNode := 4, RD_OUT_ID := "1,8,9", SD_IN_ID := "16,17,18,19,20");
        E_MERGE : E_MERGE;
        WORD2WORD_1 : WORD2WORD(IN := 2456);
        DWORD2DWORD : DWORD2DWORD(IN := 15789346);
        BYTE2BYTE_1 : BYTE2BYTE(IN := 200);
        E_CYCLE_5 : E_CYCLE(DT := T#3s);
        E_SR_3 : E_SR;
        E_SWITCH_3 : E_SWITCH;
        SINT2SINT_2 : SINT2SINT;
        INT2INT : INT2INT;
        REAL2REAL_1 : REAL2REAL;
        F_LINT_TO_LWORD : F_LINT_TO_LWORD(IN := 149486213156489);
      END_FBS
      EVENT_CONNECTIONS
        E_MERGE.EO TO a.TRANSMIT_TRG;
        a.ESD TO PUBLISH_1.REQ;
        Rx_TRG_CYC.EO TO a.SEND_RD;
        a.ESD TO E_DELAY_1.START;
        a.INITO TO PUBLISH_1.INIT;
        E_DELAY_1.EO TO E_MERGE.EI2;
        Tx_DELAY.EO TO E_MERGE.EI1;
        ROUND_CYC.EO TO a.ROUND_START;
        SUBSCRIBE_1.INITO TO a.INIT;
        ROUND_CYC.EO TO Tx_DELAY.START;
        SUBSCRIBE_1.IND TO a.REQ_RD;
        START.COLD TO ROUND_CYC.START;
        START.WARM TO ROUND_CYC.START;
        START.COLD TO E_DELAY_1.START;
        START.WARM TO E_DELAY_1.START;
        START.COLD TO Rx_TRG_CYC.START;
        START.WARM TO Rx_TRG_CYC.START;
        START.COLD TO SUBSCRIBE_1.INIT;
        START.WARM TO SUBSCRIBE_1.INIT;
        WORD2WORD_1.CNF TO a.REQ2;
        DWORD2DWORD.CNF TO a.REQ3;
        BYTE2BYTE_1.CNF TO a.REQ1;
        START.COLD TO E_CYCLE_5.START;
        START.WARM TO E_CYCLE_5.START;
        E_SR_3.EO TO BYTE2BYTE_1.REQ;
        E_SR_3.EO TO WORD2WORD_1.REQ;
        E_SR_3.EO TO DWORD2DWORD.REQ;
        E_SWITCH_3.EO1 TO E_SR_3.R;
        E_SWITCH_3.EO0 TO E_SR_3.S;
        E_CYCLE_5.EO TO E_SWITCH_3.EI;
        a.ERD TO REAL2REAL_1.REQ;
        a.ERD TO INT2INT.REQ;
        a.ERD TO SINT2SINT_2.REQ;
        E_SR_3.EO TO F_LINT_TO_LWORD.REQ;
        F_LINT_TO_LWORD.CNF TO a.REQ4;
      END_CONNECTIONS
      DATA_CONNECTIONS
        a.SD_OUT TO PUBLISH_1.SD_1;
        SUBSCRIBE_1.RD_1 TO a.RD_IN;
        WORD2WORD_1.OUT TO a.SD_IN_2;
        DWORD2DWORD.OUT TO a.SD_IN_3;
        BYTE2BYTE_1.OUT TO a.SD_IN_1;
        E_SR_3.Q TO E_SWITCH_3.G;
        a.RD_OUT_3 TO SINT2SINT_2.IN;
        a.RD_OUT_2 TO INT2INT.IN;
        a.RD_OUT_1 TO REAL2REAL_1.IN;
        F_LINT_TO_LWORD.OUT TO a.SD_IN_4;
      END_CONNECTIONS
    END_RESOURCE
  END_DEVICE
  MAPPINGS
    TestDataTypeApp.WORD2WORD_1 ON BeagleBoneBlack_3.EMB_RES.WORD2WORD_1;
    TestDataTypeApp.DWORD2DWORD ON BeagleBoneBlack_3.EMB_RES.DWORD2DWORD;
    TestDataTypeApp.BYTE2BYTE_1 ON BeagleBoneBlack_3.EMB_RES.BYTE2BYTE_1;
    TestDataTypeApp.E_CYCLE_5 ON BeagleBoneBlack_3.EMB_RES.E_CYCLE_5;
    TestDataTypeApp.E_SR_3 ON BeagleBoneBlack_3.EMB_RES.E_SR_3;
    TestDataTypeApp.E_SWITCH_3 ON BeagleBoneBlack_3.EMB_RES.E_SWITCH_3;
    TestDataTypeApp.F_MUL_3 ON BeagleBoneBlack_2.EMB_RES.F_MUL_3;
    TestDataTypeApp.INT2INT_4 ON BeagleBoneBlack_2.EMB_RES.INT2INT_4;
    TestDataTypeApp.F_ULINT_TO_LREAL ON BeagleBoneBlack.EMB_RES.F_ULINT_TO_LREAL;
    TestDataTypeApp.F_MUL_2 ON BeagleBoneBlack_2.EMB_RES.F_MUL_2;
    TestDataTypeApp.INT2INT_3 ON BeagleBoneBlack_2.EMB_RES.INT2INT_3;
    TestDataTypeApp.F_DINT_TO_ULINT ON BeagleBoneBlack_2.EMB_RES.F_DINT_TO_ULINT;
    TestDataTypeApp.F_LINT_TO_ULINT ON BeagleBoneBlack_1.EMB_RES.F_LINT_TO_ULINT;
    TestDataTypeApp.F_DINT_TO_LINT ON BeagleBoneBlack_2.EMB_RES.F_DINT_TO_LINT;
    TestDataTypeApp.WORD2WORD ON BeagleBoneBlack_1.EMB_RES.WORD2WORD;
    TestDataTypeApp.BYTE2BYTE ON BeagleBoneBlack.EMB_RES.BYTE2BYTE;
    TestDataTypeApp.INT2INT_2 ON BeagleBoneBlack_2.EMB_RES.INT2INT_2;
    TestDataTypeApp.F_MUL_1 ON BeagleBoneBlack_2.EMB_RES.F_MUL_1;
    TestDataTypeApp.E_CTU_3 ON BeagleBoneBlack_2.EMB_RES.E_CTU_3;
    TestDataTypeApp.E_PERMIT_4 ON BeagleBoneBlack_2.EMB_RES.E_PERMIT_4;
    TestDataTypeApp.E_SR_2 ON BeagleBoneBlack_2.EMB_RES.E_SR_2;
    TestDataTypeApp.E_SWITCH_2 ON BeagleBoneBlack_2.EMB_RES.E_SWITCH_2;
    TestDataTypeApp.E_CYCLE_4 ON BeagleBoneBlack_2.EMB_RES.E_CYCLE_4;
    TestDataTypeApp.F_INT_TO_SINT ON BeagleBoneBlack_1.EMB_RES.F_INT_TO_SINT;
    TestDataTypeApp.FB_CTD ON BeagleBoneBlack_1.EMB_RES.FB_CTD;
    TestDataTypeApp.UINT2UINT_2 ON BeagleBoneBlack_2.EMB_RES.UINT2UINT_2;
    TestDataTypeApp.F_MUL ON BeagleBoneBlack_2.EMB_RES.F_MUL;
    TestDataTypeApp.DINT2DINT ON BeagleBoneBlack_1.EMB_RES.DINT2DINT;
    TestDataTypeApp.UDINT2UDINT ON BeagleBoneBlack.EMB_RES.UDINT2UDINT;
    TestDataTypeApp.LREAL2LREAL_1 ON BeagleBoneBlack_2.EMB_RES.LREAL2LREAL_1;
    TestDataTypeApp.LREAL2LREAL ON BeagleBoneBlack_1.EMB_RES.LREAL2LREAL;
    TestDataTypeApp.USINT2USINT_1 ON BeagleBoneBlack.EMB_RES.USINT2USINT_1;
    TestDataTypeApp.INT2INT_1 ON BeagleBoneBlack_1.EMB_RES.INT2INT_1;
    TestDataTypeApp.SINT2SINT_2 ON BeagleBoneBlack_3.EMB_RES.SINT2SINT_2;
    TestDataTypeApp.UINT2UINT_1 ON BeagleBoneBlack.EMB_RES.UINT2UINT_1;
    TestDataTypeApp.E_CTU_2 ON BeagleBoneBlack.EMB_RES.E_CTU_2;
    TestDataTypeApp.USINT2USINT ON BeagleBoneBlack_2.EMB_RES.USINT2USINT;
    TestDataTypeApp.SINT2SINT_1 ON BeagleBoneBlack_1.EMB_RES.SINT2SINT_1;
    TestDataTypeApp.INT2INT ON BeagleBoneBlack_3.EMB_RES.INT2INT;
    TestDataTypeApp.UINT2UINT ON BeagleBoneBlack_2.EMB_RES.UINT2UINT;
    TestDataTypeApp.E_CTU_1 ON BeagleBoneBlack_1.EMB_RES.E_CTU_1;
    TestDataTypeApp.E_PERMIT_3 ON BeagleBoneBlack_1.EMB_RES.E_PERMIT_3;
    TestDataTypeApp.E_PERMIT_2 ON BeagleBoneBlack_1.EMB_RES.E_PERMIT_2;
    TestDataTypeApp.E_SR_1 ON BeagleBoneBlack_1.EMB_RES.E_SR_1;
    TestDataTypeApp.E_SWITCH_1 ON BeagleBoneBlack_1.EMB_RES.E_SWITCH_1;
    TestDataTypeApp.E_CYCLE_3 ON BeagleBoneBlack_1.EMB_RES.E_CYCLE_3;
    TestDataTypeApp.FB_RANDOM_1 ON BeagleBoneBlack_1.EMB_RES.FB_RANDOM_1;
    TestDataTypeApp.E_CYCLE_2 ON BeagleBoneBlack_1.EMB_RES.E_CYCLE_2;
    TestDataTypeApp.E_CTU ON BeagleBoneBlack.EMB_RES.E_CTU;
    TestDataTypeApp.E_PERMIT_1 ON BeagleBoneBlack.EMB_RES.E_PERMIT_1;
    TestDataTypeApp.E_PERMIT ON BeagleBoneBlack.EMB_RES.E_PERMIT;
    TestDataTypeApp.E_SR ON BeagleBoneBlack.EMB_RES.E_SR;
    TestDataTypeApp.E_SWITCH ON BeagleBoneBlack.EMB_RES.E_SWITCH;
    TestDataTypeApp.E_CYCLE_1 ON BeagleBoneBlack.EMB_RES.E_CYCLE_1;
    TestDataTypeApp.FB_RANDOM ON BeagleBoneBlack.EMB_RES.FB_RANDOM;
    TestDataTypeApp.E_CYCLE ON BeagleBoneBlack.EMB_RES.E_CYCLE;
    TestDataTypeApp.DWORD2DWORD_1 ON BeagleBoneBlack_2.EMB_RES.DWORD2DWORD_1;
    TestDataTypeApp.REAL2REAL_1 ON BeagleBoneBlack_3.EMB_RES.REAL2REAL_1;
    TestDataTypeApp.F_LWORD_TO_WORD ON BeagleBoneBlack_2.EMB_RES.F_LWORD_TO_WORD;
    TestDataTypeApp.F_LINT_TO_LWORD ON BeagleBoneBlack_3.EMB_RES.F_LINT_TO_LWORD;
  END_MAPPINGS
  SEGMENTS
    Ethernet : Ethernet;
  END_SEGMENTS
  LINKS
    BeagleBoneBlack => Ethernet;
    BeagleBoneBlack_1 => Ethernet;
    BeagleBoneBlack_2 => Ethernet;
    BeagleBoneBlack_3 => Ethernet;
  END_LINKS
END_SYSTEM
